{attribute 'enable_dynamic_creation'}
FUNCTION_BLOCK FB_DimSlot EXTENDS FB_Slot
VAR_INPUT
END_VAR
VAR_OUTPUT
END_VAR
VAR
	stDimension : ST_3DDimension;
END_VAR

PROPERTY P_rDimDepth : REAL
GET
P_rDimDepth := stDimension.Depth;
END_GET
SET
stDimension.Depth := P_rDimDepth;
END_SET
END_PROPERTY

PROPERTY P_rDimHeight : REAL
GET
P_rDimHeight := stDimension.Height;
END_GET
SET
stDimension.Height := P_rDimHeight;
END_SET
END_PROPERTY

PROPERTY P_rDimWidth : REAL
GET
P_rDimWidth := stDimension.Width;
END_GET
SET
stDimension.Width := P_rDimWidth;
END_SET
END_PROPERTY

PROPERTY P_stDimension : ST_3DDimension
GET
P_stDimension := stDimension;
END_GET
SET
stDimension := P_stDimension;
END_SET
END_PROPERTY

END_FUNCTION_BLOCK

(* stored: Version 1.1.0.1, ProductVersion 3.1.4022.18
   POU FB_DimSlot: Id {9535a7d4-4b3e-49d7-8b14-f087bc74f964}, SpecialFunc None
   Property P_rDimDepth: Id {ee63836d-51f3-40d7-9ae2-e59c48159f75}
   Get Get: Id {88584d37-7d2d-4a98-ae29-6763ff2c4c0d}
   Set Set: Id {9d4a2c1e-a3ed-4d90-9b85-448da49af184}
   Property P_rDimHeight: Id {d8c14121-9866-4520-a1fd-3a3eb85f4315}
   Get Get: Id {6966fb0e-9da7-4307-b041-9c339b580b89}
   Set Set: Id {e6593a3d-e4e0-4332-9e75-25a595f14ae0}
   Property P_rDimWidth: Id {8fe2505e-8eaa-4179-bb39-da70899792ce}
   Get Get: Id {b88113c2-2e54-47d6-bacc-77516cbb2f8d}
   Set Set: Id {5d7a347f-fcae-4c89-943d-5cd7fd03cef3}
   Property P_stDimension: Id {4ce14945-dc41-4e8a-9124-7a51ccdca2a8}
   Get Get: Id {54b01c9b-38f2-4e9a-93ff-b6e3b467755b}
   Set Set: Id {3321d9c1-2193-46fa-98ca-43a12042e4de} *)
